// TIA Portal V17 export
// export: Created 2024-10-17T14:16:17.5295494Z, ExportSetting WithDefaults, DisplayName Totally Integrated Automation Portal, DisplayVersion V17 Update 4, DisplayName TIA Portal Openness, DisplayVersion V17 Update 4, DisplayName TIA Portal Version Control Interface, DisplayVersion V17, DisplayName SINAMICS Startdrive Advanced, DisplayVersion V17 Update2, DisplayName SINAMICS Startdrive G130, G150, S120, S150, SINAMICS MV, S210, DisplayVersion V17 Update2, DisplayName SINAMICS Startdrive G110M, G120, G120C, G120D, G120P, G115D, DisplayVersion V17 Update2, DisplayName STEP 7 Professional, DisplayVersion V17 Update 4, DisplayName STEP 7 Safety, DisplayVersion V17, DisplayName WinCC Advanced / Unified PC, DisplayVersion V17 Update 4
TYPE "LPMLV2022_typeCumulativeTimes"
TITLE = LPMLV2022_typeCumulativeTimes
// Support: tech.team.motioncontrol@siemens.com
// stored: IsFailsafeCompliant false
   STRUCT
      AccTimeSinceReset { ExternalWritable := 'False'} : DInt;   // Accumulated Time Since Last Reset. The tag represents the amount of time (in seconds) since the reset has been triggered for a particular collection of cumulative times. When a reset for a particular collection is triggered, all times inside the structure for that collection are reset
      ModeStateTimes { ExternalWritable := 'False'} : Array[0.."LPMLV2022_ADMIN_NUMBER_OF_MODES_UPPER_LIM"] of "LPMLV2022_typeModeStateTimes";   // Structured Array of Mode and State Time Values for each Cumulative Time Tracker. This tag is a collection of times for modes and states since the last timer reset was executed
   END_STRUCT;
END_TYPE
